FUNCTION_BLOCK FileBasedByteBuffer IMPLEMENTS I_Buffer
VAR
	
	fileName : STRING;
	state: (IDLE, START_WRITING, INITIALISE, CYCLIC_WRITE, CLOSE) := IDLE;
	binaryFileWriter : ByteBufferFileWriter('');
		
	buffer1 : ARRAY [0..GVL_ByteBufferConstants.FILE_WRITE_BUFFER_SIZE] OF BYTE;
	buffer2 : ARRAY [0..GVL_ByteBufferConstants.FILE_WRITE_BUFFER_SIZE] OF BYTE;
	byteBuffer1 : ByteBuffer(ADR(buffer1),SIZEOF(buffer1));
	byteBuffer2 : ByteBuffer(ADR(buffer2),SIZEOF(buffer2));
	
	currentlySavingBuffer : I_Buffer := byteBuffer2;
	standbyBuffer : I_Buffer := byteBuffer2;
	activeBuffer : I_Buffer := byteBuffer1;
	
END_VAR

CASE state OF
		
	IDLE: //
	
	START_WRITING: 
	
		byteBuffer1.Reset();
		byteBuffer2.Reset();
		
		activeBuffer := byteBuffer1;
		standbyBuffer := byteBuffer2;
		currentlySavingBuffer := standbyBuffer;
		
		binaryFileWriter.OpenFile(fileName);
		state := CYCLIC_WRITE;
		
	CYCLIC_WRITE: //
		
	CLOSE: 
	
		IF activeBuffer.Size = 0 AND standbyBuffer.Size = 0 THEN
			IF binaryFileWriter.CloseFile() THEN 
				state := IDLE;
			END_IF
		END_IF
	
END_CASE

binaryFileWriter();

IF binaryFileWriter.WriteComplete THEN
	currentlySavingBuffer.Reset();
END_IF

IF standbyBuffer.Size = 0 THEN
	IF binaryFileWriter.WriteByteBufferToFile(activeBuffer) THEN
		currentlySavingBuffer := activeBuffer;
		activeBuffer := standbyBuffer;
		standbyBuffer := currentlySavingBuffer;
	END_IF
END_IF

METHOD PUBLIC AddBoolToBuffer : BOOL
VAR_IN_OUT
	Field : BOOL;
END_VAR
AddBoolToBuffer := activeBuffer.AddBoolToBuffer(Field);
END_METHOD

METHOD PUBLIC AddCharToBuffer : BOOL
VAR_IN_OUT
	Field : BYTE;
END_VAR
AddCharToBuffer := activeBuffer.AddCharToBuffer(Field);
END_METHOD

METHOD PUBLIC AddIntToBuffer : BOOL
VAR_IN_OUT
	Field : INT;
END_VAR
AddIntToBuffer := activeBuffer.AddIntToBuffer(Field);
END_METHOD

PROPERTY PUBLIC Address : pointer to byte
GET
Address := activeBuffer.Address;
END_GET
END_PROPERTY

METHOD PUBLIC AddStringToBuffer : BOOL
VAR_IN_OUT
	stringToWrite : STRING;
END_VAR
AddStringToBuffer := activeBuffer.AddStringToBuffer(stringToWrite);
END_METHOD

PROPERTY PUBLIC IsActive : BOOL
GET
IsActive := state = CYCLIC_WRITE;
END_GET
END_PROPERTY

PROPERTY PUBLIC IsStopped : BOOL
GET
IsStopped := state = IDLE;
END_GET
END_PROPERTY

PROPERTY PUBLIC Remaining : UDINT
GET
Remaining := activeBuffer.Remaining;
END_GET
END_PROPERTY

METHOD Reset
VAR_INPUT
END_VAR
activeBuffer.Reset();
END_METHOD

PROPERTY PUBLIC Size : udint
GET
Size := activeBuffer.Size;
END_GET
END_PROPERTY

METHOD PUBLIC Start : BOOL
VAR_INPUT
	fileName : STRING;
END_VAR
IF State = IDLE THEN
	THIS^.fileName := fileName;
	State := START_WRITING;
	Start := TRUE;
END_IF
END_METHOD

METHOD PUBLIC Stop : BOOL
VAR_INPUT
END_VAR
IF State = CYCLIC_WRITE THEN
	State := CLOSE;
	Stop := TRUE;
END_IF
END_METHOD

END_FUNCTION_BLOCK

(* stored: Version 1.1.0.1, ProductVersion 3.1.4024.4
   POU FileBasedByteBuffer: Id {fd1e91c2-96b3-4851-9be2-08b665937ee6}, SpecialFunc None
   Method AddBoolToBuffer: Id {b97dca57-dc88-4275-b896-2c93500eacb5}
   Method AddCharToBuffer: Id {abbadc54-ab7d-4cdd-a01c-7a6150c9e78b}
   Method AddIntToBuffer: Id {22daea51-e3a6-44fb-927e-bfe128106c4d}
   Property Address: Id {4d29680e-eb35-4d46-9e04-dec0dcc8a1ce}
   Get Get: Id {05fd5825-3c51-43b6-8acb-b3f5e57abcd1}
   Method AddStringToBuffer: Id {14795828-7035-49b9-a533-783abaf0e2a8}
   Property IsActive: Id {e3523571-9469-4ad4-93c1-782fe8ab88ef}
   Get Get: Id {db4f71f0-98ea-4e81-a7fe-50180cc1d8c6}
   Property IsStopped: Id {bf6af49b-19cf-4f33-ad0d-85437c531d29}
   Get Get: Id {7e61e412-a2da-4323-8e85-feebe10450fd}
   Property Remaining: Id {268fc45e-1b26-4c9a-8f5d-e6eac4b9d8b6}
   Get Get: Id {27c1fb4d-b9b2-4d9e-8e19-60c793458ef8}
   Method Reset: Id {48a32e79-a26c-47a5-ab47-fd7f2dd067be}
   Property Size: Id {41868a1a-854c-4fc4-9a99-65a01352797c}
   Get Get: Id {cbfd5190-ee38-4a3c-b56c-2a2c94733cd7}
   Method Start: Id {011f7e44-5747-47a2-8dfe-0eb0e68b9580}
   Method Stop: Id {20754d56-1d9d-40df-9eb2-0c386c403ad6} *)
